TYPE ST_SCANNER_ManualStatus :
STRUCT
	bConfigure			: BOOL;	
	bBrowseLive			: BOOL;	
	bBrowseDiag			: BOOL;
END_STRUCT
END_TYPE

(* stored: Version 1.1.0.1
   DUT ST_SCANNER_ManualStatus: Id {3c5459d2-a8f8-4cae-b088-4153bc272cac} *)
